TYPE ST_InputsLiftTable :
STRUCT
	HW		: ST_HW_InputsLiftTable; //Hardware inputs
END_STRUCT
END_TYPE

(* stored: Version 1.1.0.1, ProductVersion 3.1.4024.9
   DUT ST_InputsLiftTable: Id {c94b01a8-c264-4933-a04c-13a14731bcb7} *)
